INTERFACE I_MarkDefinition

(*
  Get a mark definition.
  nIdx= 1.._nMarks = registered marks
  nIdx= 0 - selects last mark 
  nIdx=-1 - selects boarder mark
*)
METHOD getMark : POINTER TO ST_MarkDefinition
VAR_INPUT
  nIdx : DINT; // mark index: 1.._nMarks, 0 = last (endMark) 
END_VAR
END_METHOD

(*Number of registered marks*)
PROPERTY nMarks : UDINT
GET
END_GET
END_PROPERTY

(*Number of detected marks*)
PROPERTY nMarksDetected : UDINT
GET
END_GET
END_PROPERTY

(*
  Reset all registered marks
*)
METHOD ResetMarkStates
END_METHOD

METHOD saveMark : BOOL
VAR_INPUT
  pMark : POINTER TO ST_MarkDefinition;
END_VAR
END_METHOD

END_INTERFACE

(* stored: Version 1.1.0.1, ProductVersion 3.1.4024.11
   Itf I_MarkDefinition: Id {f4a29f8c-4eaf-41ce-b828-08db2ca8315b}
   Method getMark: Id {a705d2a4-440b-4c23-aa2d-20beb49f17b2}
   Property nMarks: Id {a84bd018-75eb-48e2-9072-e404c7a08399}
   Get Get: Id {c46ec7e9-ad3c-40e2-b627-61438f9d581d}
   Property nMarksDetected: Id {7be5b84f-a5c2-4e6c-82ab-47a30715665a}
   Get Get: Id {d8e77488-d20e-400e-a298-b5b213453b01}
   Method ResetMarkStates: Id {96e195a2-f992-484c-b0ec-49ab27b40bd3}
   Method saveMark: Id {db84adae-9689-45fe-ab25-5ab7f86f89e2} *)
